// TIA Portal V19 export
FUNCTION "Block_1" : Void   // FC1, FBD
TITLE = FC
{ S7_Optimized_Access := 'TRUE' }
// stored: SetENOAutomatically false
   VAR_INPUT
      in : Bool;
   END_VAR
   VAR_OUTPUT
      out : Bool;
   END_VAR
BEGIN

REGION Network 1: network1
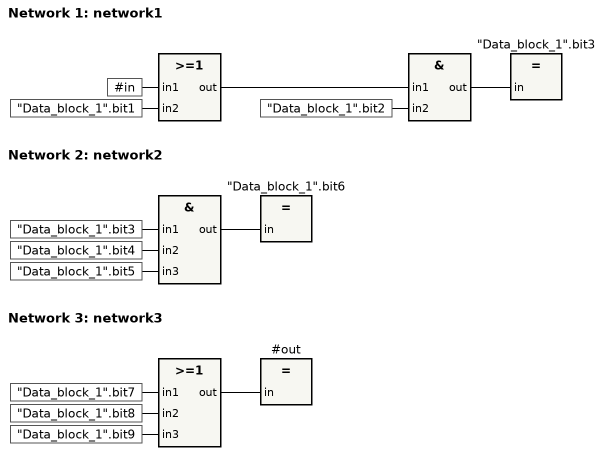
   "Data_block_1".bit3 := (#in OR "Data_block_1".bit1) AND "Data_block_1".bit2;
END_REGION

REGION Network 2: network2
   "Data_block_1".bit6 := "Data_block_1".bit3 AND "Data_block_1".bit4 AND "Data_block_1".bit5;
END_REGION

REGION Network 3: network3
   #out := "Data_block_1".bit7 OR "Data_block_1".bit8 OR "Data_block_1".bit9;
END_REGION
END_FUNCTION
